FUNCTION_BLOCK CheckStatus
VAR_INPUT
	F_Reset: BOOL;
	Data: ARRAY [1..100] OF BOOL;
END_VAR
VAR_OUTPUT
	Status: BOOL;
	Reset : R_TRIG;
END_VAR
VAR
	i: UINT;
	j: UINT;
	
	a: UINT;
	
	SeqCheck: ARRAY [1..300] OF UINT;
	CheckReset: BOOL;
	SeqIndex: INT;
END_VAR

(* new Management Error *)
CASE SeqIndex OF 
	0: 
		FOR i:=1 TO 100 BY 1 DO //program for ini bertujuan untuk mengiterasi i dari 1 sampai 100
			IF Data[i] THEN		//jika pada iterasi Data terdapat nilai ke-i = true
				Status:=TRUE;   //maka output status menjadi true
				j := 0;         //dan index j = 0
				i := 100;       //dan index i = 100
				seqIndex := 10; //SeqIndex berpindah ke 10
			END_IF
			
		END_FOR
	10: 
		Reset( CLK := F_Reset);               //Raising Trigger/Trigger Positif didapat oleh F_Reset, maka reset akan aktif
		IF Reset.Q AND NOT CheckReset THEN    //jika reset bernilai TRUE dan CheckReset bernilai FALSE, maka:
			i := 0;                           //index = 0
			CheckReset:=TRUE;                 //CheckReset = TRUE
			seqIndex := 20;                   //SeqIndex berpindah ke sequence 20
		END_IF
	20: 
		IF CheckReset THEN 
			FOR j:=1 TO 100 BY 1 DO           //iterasikan j dari 1 sampai dengan 100
				IF NOT Data[j] THEN		      //jika dalam array data J terdapoat nilai TRUE
					Status:=FALSE;            //Status jadi False
					CheckReset:=FALSE;        //CheckReset jadi False
					j := 100 ;                //J berubah index ke 100
					seqIndex := 0;            //SeqIndex berubah ke keadaan awal
				END_IF
			END_FOR
		END_IF 
END_CASE
(* old management error *problem Delay Respons
IF CheckReset THEN
	CASE SeqCheck[a] OF
		0:
			IF NOT Data[a] THEN
				SeqCheck[a]:=10;
			ELSE
				CheckReset:=FALSE;
			END_IF
		10:
			IF a = 300 THEN
				Status:=FALSE;
				CheckReset:=FALSE;
			ELSE
				a := a + 1;
			END_IF
	END_CASE
ELSE
	FOR j:=1 TO 300 BY 1 DO
		SeqCheck[j]:=0;
	END_FOR
	a:=1;
END_IF

*)

END_FUNCTION_BLOCK

(* stored: Version 1.1.0.1, ProductVersion 3.1.4024.6
   POU CheckStatus: Id {5fe12cb5-a914-4bcc-971d-fff763150b3c}, SpecialFunc None *)
